(* PLC project  *)

PROGRAM P
  VAR  (* added by the conversion: wires and edge detectors of the diagram *)
    _OR3_OUT : BOOL;
  END_VAR

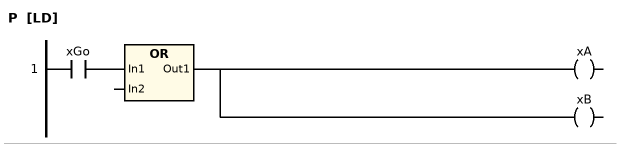
(* LD diagram, written out as Structured Text *)
_OR3_OUT := OR(In1 := xGo);
xA := _OR3_OUT;
xB := _OR3_OUT;
END_PROGRAM
